TYPE M3IOStatuses :
STRUCT
	///Is the I/O in a healthy state?
	healthStatus: HealthStatus;
END_STRUCT
END_TYPE

(* stored: Version 1.1.0.1, ProductVersion 3.1.4019.2
   DUT M3IOStatuses: Id {4a13338f-a1c6-4d77-8bc8-511e4af1c31b} *)
